TYPE stBH0HPL_Line EXTENDS stPIM_LineEventsModule :
STRUCT

	{attribute 'OPC.UA.DA' := '1'}
	stStation_BH0HPL01 : stPIM_StationEventsModule_3_Machine;
END_STRUCT
END_TYPE

(* stored: Version 1.1.0.1, ProductVersion 3.1.4024.15
   DUT stBH0HPL_Line: Id {67a7ccbc-9bfd-458f-a6cc-73f626a83089} *)
